// TIA Portal V15.1 export
// export: Created 2020-06-12T07:35:49.6787109Z, ExportSetting None, DisplayName Totally Integrated Automation Portal, DisplayVersion V15.1, DisplayName TIA Portal Openness, DisplayVersion V15.1, DisplayName STEP 7 Professional, DisplayVersion V15.1, DisplayName STEP 7 Safety, DisplayVersion V15.1, DisplayName WinCC Advanced, DisplayVersion V15.1
FUNCTION "MELT_Meas_Energy" : Void   // FC111, FBD
{ S7_Optimized_Access := 'TRUE' }
// stored: SetENOAutomatically False
   VAR_TEMP
      _reset : Bool;
      _imp : Bool;
      _factor : Real;
   END_VAR
BEGIN

REGION Network 1: Reset counters
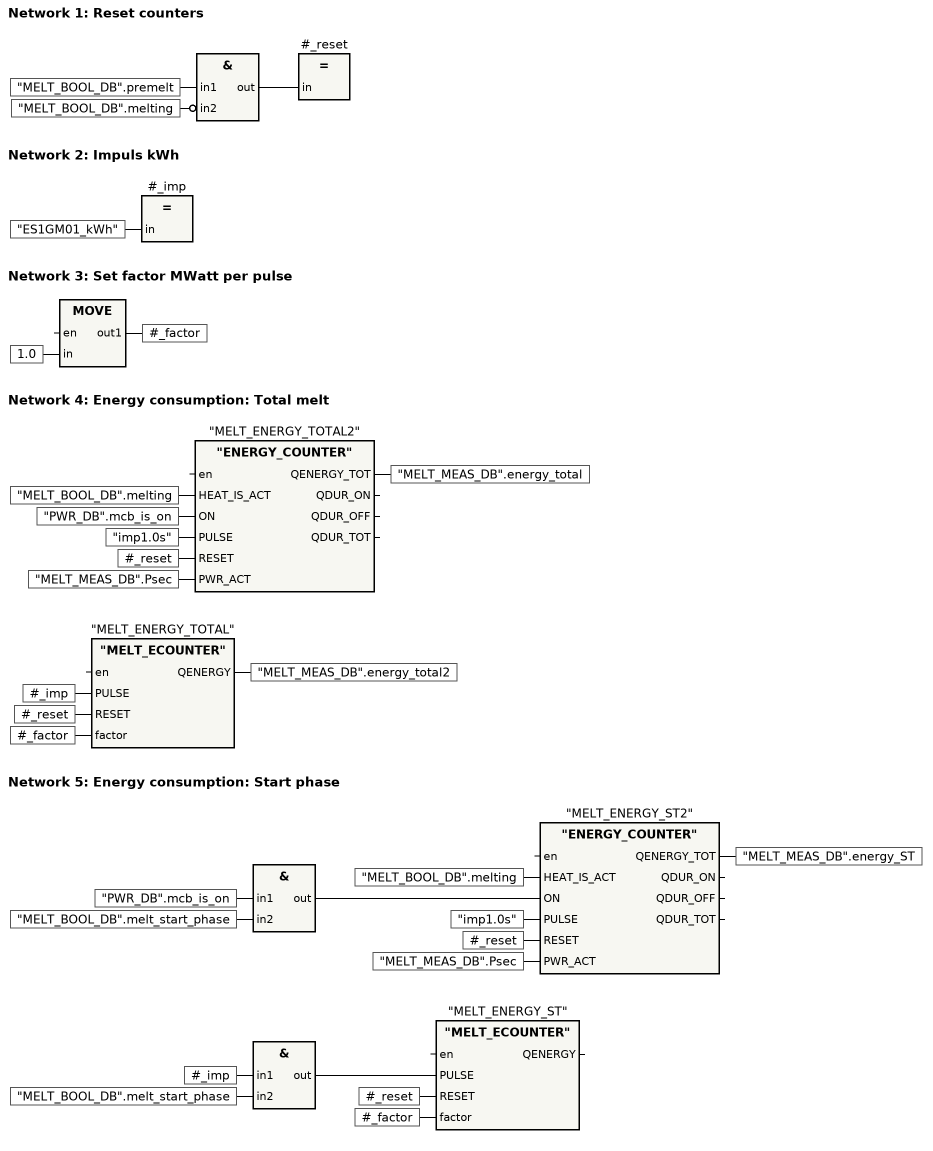
   #_reset := "MELT_BOOL_DB".premelt AND NOT "MELT_BOOL_DB".melting;
END_REGION

REGION Network 2: Impuls kWh
   #_imp := "ES1GM01_kWh";
END_REGION

REGION Network 3: Set factor MWatt per pulse
   #_factor := 1.0;
END_REGION

REGION Network 4: Energy consumption: Total melt
   // "IO_ESMLS1".XS01_pwr_pls
   "MELT_ENERGY_TOTAL2"(HEAT_IS_ACT := "MELT_BOOL_DB".melting,   // "ENERGY_COUNTER"
                        ON := "PWR_DB".mcb_is_on,
                        PULSE := "imp1.0s",
                        RESET := #_reset,
                        PWR_ACT := "MELT_MEAS_DB".Psec,
                        QENERGY_TOT => "MELT_MEAS_DB".energy_total);
   "MELT_ENERGY_TOTAL"(PULSE := #_imp,   // "MELT_ECOUNTER"
                       RESET := #_reset,
                       factor := #_factor,
                       QENERGY => "MELT_MEAS_DB".energy_total2);
END_REGION

REGION Network 5: Energy consumption: Start phase
   // "IO_ESMLS1".XS01_pwr_pls
   "MELT_ENERGY_ST2"(HEAT_IS_ACT := "MELT_BOOL_DB".melting,   // "ENERGY_COUNTER"
                     ON := "PWR_DB".mcb_is_on AND "MELT_BOOL_DB".melt_start_phase,
                     PULSE := "imp1.0s",
                     RESET := #_reset,
                     PWR_ACT := "MELT_MEAS_DB".Psec,
                     QENERGY_TOT => "MELT_MEAS_DB".energy_ST);
   "MELT_ENERGY_ST"(PULSE := #_imp AND "MELT_BOOL_DB".melt_start_phase, RESET := #_reset, factor := #_factor);   // "MELT_ECOUNTER"
END_REGION

REGION Network 6: Energy consumption: Melt phase
   // "IO_ESMLS1".XS01_pwr_pls
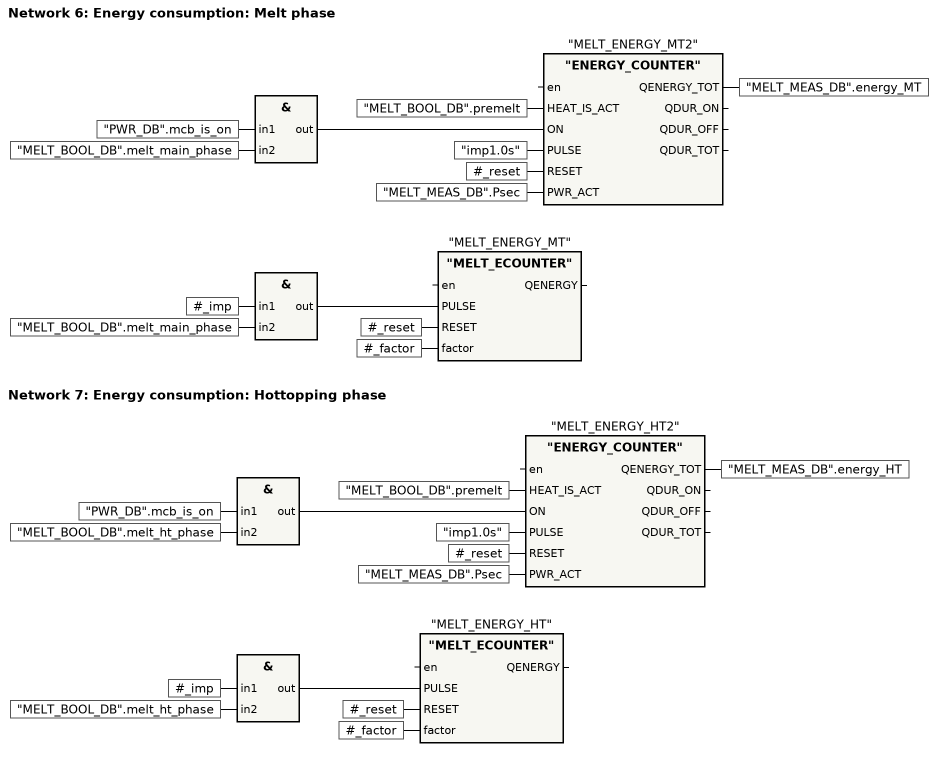
   "MELT_ENERGY_MT2"(HEAT_IS_ACT := "MELT_BOOL_DB".premelt,   // "ENERGY_COUNTER"
                     ON := "PWR_DB".mcb_is_on AND "MELT_BOOL_DB".melt_main_phase,
                     PULSE := "imp1.0s",
                     RESET := #_reset,
                     PWR_ACT := "MELT_MEAS_DB".Psec,
                     QENERGY_TOT => "MELT_MEAS_DB".energy_MT);
   "MELT_ENERGY_MT"(PULSE := #_imp AND "MELT_BOOL_DB".melt_main_phase, RESET := #_reset, factor := #_factor);   // "MELT_ECOUNTER"
END_REGION

REGION Network 7: Energy consumption: Hottopping phase
   // "IO_ESMLS1".XS01_pwr_pls
   "MELT_ENERGY_HT2"(HEAT_IS_ACT := "MELT_BOOL_DB".premelt,   // "ENERGY_COUNTER"
                     ON := "PWR_DB".mcb_is_on AND "MELT_BOOL_DB".melt_ht_phase,
                     PULSE := "imp1.0s",
                     RESET := #_reset,
                     PWR_ACT := "MELT_MEAS_DB".Psec,
                     QENERGY_TOT => "MELT_MEAS_DB".energy_HT);
   "MELT_ENERGY_HT"(PULSE := #_imp AND "MELT_BOOL_DB".melt_ht_phase, RESET := #_reset, factor := #_factor);   // "MELT_ECOUNTER"
END_REGION

REGION Network 8 (SCL): Energy consumption [kWh/t]
   "MELT_MEAS_DB".kWhT := 1000.0 * "MELT_MEAS_DB".energy_total / "MELT_MEAS_DB".ingot_weight;
END_REGION
END_FUNCTION
